{attribute 'qualified_only'}
TYPE ENUM_ATM_States :
(
    Unknown := 0,
    OUT := 1,
    TARGET1 := 2,
    TARGET2 := 3,
    TARGET3 := 4,
    TARGET4 := 5,
    TARGET5 := 6
);
END_TYPE

(* stored: Version 1.1.0.1
   DUT ENUM_ATM_States: Id {39e72780-ebe1-47a1-93c3-70f8a4ded457} *)
